FUNCTION_BLOCK FB_HexDecoder
VAR_INPUT
END_VAR
VAR_OUTPUT
END_VAR
VAR
END_VAR

END_FUNCTION_BLOCK

(* stored: Version 1.1.0.1
   POU FB_HexDecoder: Id {433cdd27-5eab-439a-84f2-623599003218}, SpecialFunc None *)
